TYPE ZDataRecipe :
STRUCT
  RecipeParam1 : LREAL;
  RecipeParam2 : LREAL;
  RecipeParam3 : LREAL;
END_STRUCT
END_TYPE

(* stored: Version 1.1.0.1
   DUT ZDataRecipe: Id {2c776f8c-cc7c-4169-af84-9e4ea901d0d7} *)
